// TIA Portal V19 export
FUNCTION_BLOCK "Pu_Versorgung.GP0x"   // FB1010, LAD
{ S7_Optimized_Access := 'TRUE' }
// Funktionen:  HF Versorgung  / Spülen
// stored: AutoNumber false, MemoryReserve 100, SetENOAutomatically false
   VAR RETAIN
      In { ExternalVisible := 'False'; ExternalWritable := 'False'} : Struct
         Auto : Bool;   // Paneltaste
         Ein : Bool;   // Paneltaste
         Not_Halt : Bool;
         Quitt_Al_Dfl : Bool;
         kein_Gas_Alarm : Bool;
         Leckage_Pumpe_ok : Bool;
         Leckage_PFA_Uebergang_ok : Bool;
         Leckage_Doppelrohr_ok : Bool;
         Leckage_Uml_Tunnel_ok : Bool;
         Leckage_Doppelschlauch_ok : Bool;
         Niv_min : Bool;
         Niv_max : Bool;
         Niv_Min_CM01 : Bool;
         Niv_Max_CM01 : Bool;
         Niv_Übervoll_CM01 : Bool;
         Niv_Min_CM02 : Bool;
         Niv_Max_CM02 : Bool;
         Niv_Übervoll_CM02 : Bool;
         Frg_Niv_CM05 : Bool;
         SRM_Saugseite_auf : Bool;
         SRM_Saugseite_zu : Bool;
         SRM_Druckseite_auf : Bool;
         SRM_Druckseite_zu : Bool;
         SRM_Eingang_Spülltg_auf : Bool;
         SRM_Eingang_Spülltg_zu : Bool;
         SRM_Ausgang_Spülltg_auf : Bool;
         SRM_Ausgang_Spülltg_zu : Bool;
         SRM_Versogung_UV01_auf : Bool;
         SRM_Versogung_UV01_zu : Bool;
         SRM_UV01_CM01_auf : Bool;
         SRM_UV01_CM01_zu { ExternalAccessible := 'False'} : Bool;
         SRM_UV01_CM02_auf { ExternalAccessible := 'False'} : Bool;
         SRM_UV01_CM02_zu { ExternalAccessible := 'False'} : Bool;
         Anf_HF_CM01 { ExternalAccessible := 'False'} : Bool;
         Anf_HF_CM02 { ExternalAccessible := 'False'} : Bool;
         IBC_vorhanden { ExternalAccessible := 'False'} : Bool;
         Tuer_vorn_zu { ExternalAccessible := 'False'} : Bool;
         Tuer_seitlich_zu { ExternalAccessible := 'False'} : Bool;
         Imp_Dfl { ExternalAccessible := 'False'} : Bool;
         GW_Dfl { ExternalAccessible := 'False'} : Bool;
         Betriebsart { ExternalAccessible := 'False'} : USInt := 0;   // Paneltaste
         Niveau { ExternalAccessible := 'False'} : USInt;
         Dfl { ExternalAccessible := 'False'} : Real;
      END_STRUCT;
      Param { ExternalAccessible := 'False'; ExternalVisible := 'False'; ExternalWritable := 'False'} : Struct
         Spülzeit : Time;
      END_STRUCT;
      Zst { ExternalAccessible := 'False'; ExternalVisible := 'False'; ExternalWritable := 'False'} : Struct
         Niveau : USInt;
         Status_GP0x : USInt;
         Restzeit_Spülen : Time;
         Spuelen : Bool;
         Pumpen : Bool;
         Weg_frei : Bool;
         Spuelen_aktiv : Bool;
         Bedienung_erlaubt : Bool;
      END_STRUCT;
      Mld { ExternalVisible := 'False'; ExternalWritable := 'False'} : Struct
         Leckage_Pumpe : Bool;
         Leckage_PFA_Uebergang : Bool;
         Leckage_Doppelrohr : Bool;
         Leckage_Uml_Tunnel : Bool;
         Leckage_Doppelschlauch : Bool;
         Niv_Sensorfehler : Bool;
         GW_Dfl : Bool;
         UeW_Dfl_Dos : Bool;
         Leermeldung : Bool;
         Vollmeldung : Bool;
         n_Auto : Bool;
         Radarsonde_niO : Bool;
      END_STRUCT;
      Out { ExternalVisible := 'False'; ExternalWritable := 'False'} : Struct
         GP0x_Ein : Bool;
         Spülventil_Eingang : Bool;
         Spülventil_Ausgang : Bool;
         Ventil_Saugseite : Bool;
         Ventil_Druckseite : Bool;
         Ventil_Entsorgung : Bool;
         Versorgung_UV01 : Bool;
         UV01_CM01 : Bool;
         UV01_CM02 : Bool;
      END_STRUCT;
   END_VAR
   VAR
      IEC_Timer : Struct
         GW_Dfl { ExternalAccessible := 'False'; ExternalVisible := 'False'; ExternalWritable := 'False'; S7_SetPoint := 'True'} : TON_TIME;
         Spülen { S7_SetPoint := 'True'} : TP_TIME;
         Verz_Min { S7_SetPoint := 'True'} : TON_TIME;
         Imp_Dfl { S7_SetPoint := 'True'} : TON_TIME;
         Spülventil_Ausgang { S7_SetPoint := 'True'} : TOF_TIME;
         Verz_NivMax { S7_SetPoint := 'True'} : TON_TIME;
      END_STRUCT;
      R_TRIG_Hand_EIN { S7_SetPoint := 'True'} : R_TRIG;
   END_VAR
   VAR_TEMP
      Spülzeit : Time;
      posFl_Hand : Bool;
      Leckage_Versorgung_ok : Bool;
      Alarm_Dfl_Dos : Bool;
   END_VAR
   VAR CONSTANT
      Niv_TLS : USInt := 2;
      Niv_Min : USInt := 20;
      Niv_max : USInt := 90;
      Zeit_Ventil_auf : Time := T#5s;
   END_VAR
BEGIN

REGION Network 1 (SCL): Input
   // Panelbedienung und Sensoren --> Input()

   // positive Flanke "Hand Ein"
   #R_TRIG_Hand_EIN(CLK := #In.Ein,
                    Q => #posFl_Hand);
   // Freigabe Not-Halt Pumpen
   #In.Not_Halt := NOT "DB_PNOZ_IN_Out".In.NH_Frg_Pumpen OR NOT "E_Frg_AbLW";

   // Leckage Versorgung
   #Leckage_Versorgung_ok := #In.Leckage_Doppelrohr_ok AND #In.Leckage_PFA_Uebergang_ok AND #In.Leckage_Uml_Tunnel_ok AND #In.Leckage_Doppelschlauch_ok;

   // Quittierung Alarm Durchfluss
   IF #In.Quitt_Al_Dfl AND #Mld.UeW_Dfl_Dos THEN
       #Mld.UeW_Dfl_Dos := FALSE;
   END_IF;
END_REGION

REGION Network 2 (SCL): Ansteuerung
   // Alles AUS
   IF (#In.Betriebsart = 3) AND #In.Tuer_vorn_zu AND #In.Tuer_seitlich_zu AND NOT #In.Not_Halt THEN // Spülen
       // Ausschaltverzögert - Druckabbau
       #IEC_Timer.Spülventil_Ausgang(IN := #Out.Spülventil_Eingang,
                                     PT := T#3s,
                                     Q => #Out.Spülventil_Ausgang);
   ELSE
       #Out.Spülventil_Eingang := FALSE;
       #Out.Spülventil_Ausgang := FALSE;
   END_IF;

   #Zst.Restzeit_Spülen := T#0s;
   #Out.Ventil_Saugseite := FALSE;
   #Out.Ventil_Druckseite := FALSE;
   #Out.Versorgung_UV01 := FALSE;
   #Out.UV01_CM01 := FALSE;
   #Out.UV01_CM02 := FALSE;
   #Out.Ventil_Entsorgung := FALSE;
   #Out.GP0x_Ein := FALSE;

   IF #In.Tuer_vorn_zu AND #In.Tuer_seitlich_zu AND NOT #In.Not_Halt THEN
       CASE #In.Betriebsart OF
           0:  // Versorgung Auto

               // Ventile öffnen
               IF #Leckage_Versorgung_ok AND #In.kein_Gas_Alarm THEN
                   #Out.Ventil_Saugseite := #Out.Ventil_Druckseite := #Out.Versorgung_UV01 := #In.Auto;
                   #Out.UV01_CM01 := #In.Anf_HF_CM01 AND #In.Auto;
                   #Out.UV01_CM02 := #In.Anf_HF_CM02 AND #In.Auto;
               END_IF;

               // Check weg
               #Zst.Weg_frei := #In.SRM_Ausgang_Spülltg_zu AND #In.SRM_Eingang_Spülltg_zu AND
               #In.SRM_Druckseite_auf AND #In.SRM_Saugseite_auf AND #In.SRM_Versogung_UV01_auf AND
               ((#In.SRM_UV01_CM01_auf AND #In.SRM_UV01_CM02_zu AND #In.Anf_HF_CM01) OR (#In.SRM_UV01_CM02_auf AND #In.SRM_UV01_CM01_zu AND #In.Anf_HF_CM02));

               // Weg frei, Behälter nicht leer und Ziel nicht übervoll
               #Zst.Pumpen := #Zst.Weg_frei AND NOT #Mld.Leermeldung AND #In.IBC_vorhanden AND NOT #Mld.UeW_Dfl_Dos AND
               ((#In.Anf_HF_CM01 AND NOT #In.Niv_Übervoll_CM01 AND NOT #In.Niv_Max_CM01) OR (#In.Anf_HF_CM02 AND NOT #In.Niv_Übervoll_CM02 AND NOT #In.Niv_Max_CM02));

           1:  // Versorgung CM01 Hand
               // Ventile öffnen
               IF #Leckage_Versorgung_ok AND #In.kein_Gas_Alarm THEN
                   #Out.Ventil_Saugseite := #Out.Ventil_Druckseite := #Out.Versorgung_UV01 := #Out.UV01_CM01 := #In.Ein;
               END_IF;

               // Check weg
               #Zst.Weg_frei := #In.SRM_Ausgang_Spülltg_zu AND #In.SRM_Eingang_Spülltg_zu AND
               #In.SRM_Druckseite_auf AND #In.SRM_Saugseite_auf AND
               #In.SRM_Versogung_UV01_auf AND #In.SRM_UV01_CM01_auf AND #In.SRM_UV01_CM02_zu;

               // Weg frei, Behälter nicht leer und Ziel nicht übervoll
               #Zst.Pumpen := #Zst.Weg_frei AND NOT #Mld.Leermeldung AND #In.IBC_vorhanden AND NOT #In.Niv_Übervoll_CM01 AND NOT #In.Niv_Max_CM01 AND NOT #In.Niv_Min_CM01;

           2:  // Versorgung CM02 Hand
               // Ventile öffnen
               IF #Leckage_Versorgung_ok AND #In.kein_Gas_Alarm THEN
                   #Out.Ventil_Saugseite := #Out.Ventil_Druckseite := #Out.Versorgung_UV01 := #Out.UV01_CM02 := #In.Ein;
               END_IF;

               // Check Weg
               #Zst.Weg_frei := #In.SRM_Ausgang_Spülltg_zu AND #In.SRM_Eingang_Spülltg_zu AND
               #In.SRM_Druckseite_auf AND #In.SRM_Saugseite_auf AND
               #In.SRM_Versogung_UV01_auf AND #In.SRM_UV01_CM02_auf AND #In.SRM_UV01_CM01_zu;

               // Weg frei, Behälter nicht leer und Ziel nicht übervoll
               #Zst.Pumpen := #Zst.Weg_frei AND NOT #Mld.Leermeldung AND #In.IBC_vorhanden AND NOT #In.Niv_Übervoll_CM02 AND NOT #In.Niv_Max_CM02 AND NOT #In.Niv_Min_CM02;

           3: // Spülen - nur Hand
               #Zst.Pumpen := FALSE;

               IF #In.Ein THEN
                   IF #posFl_Hand THEN
                       #Zst.Spuelen_aktiv := TRUE;
                   END_IF;
                   #Out.Spülventil_Eingang := #In.Frg_Niv_CM05 AND #In.SRM_Saugseite_zu AND #In.SRM_Druckseite_zu AND #Zst.Spuelen_aktiv;

                   #IEC_Timer.Spülen(IN := #In.SRM_Eingang_Spülltg_auf AND #In.SRM_Ausgang_Spülltg_auf,
                                     PT := #Param.Spülzeit,
                                     Q => #Zst.Spuelen,
                                     ET => #Spülzeit);
                   #Zst.Restzeit_Spülen := #Param.Spülzeit - #Spülzeit;

                   IF #In.SRM_Eingang_Spülltg_auf AND #In.SRM_Ausgang_Spülltg_auf AND #In.SRM_Saugseite_zu AND #In.SRM_Druckseite_zu
                       AND NOT #Zst.Spuelen AND #Zst.Spuelen_aktiv THEN
                       #Zst.Spuelen_aktiv := FALSE;
                       #Out.Spülventil_Eingang := FALSE;
                   END_IF;

               ELSE
                   #Out.Spülventil_Eingang := FALSE;
                   #Out.Spülventil_Ausgang := FALSE;
                   #Zst.Spuelen := FALSE;
                   #Zst.Spuelen_aktiv := FALSE;
               END_IF;

           4: // Entsorgung
               #Zst.Spuelen := FALSE;
               #Zst.Pumpen := FALSE;

               //Quick Connect Entsorgung
               #Out.Ventil_Entsorgung := NOT #In.Niv_max AND (#In.Niveau < 85) AND #In.IBC_vorhanden;

       END_CASE;
       // Pumpe an 
       #Out.GP0x_Ein := #Zst.Pumpen AND #In.Leckage_Pumpe_ok;
   END_IF;
END_REGION

REGION Network 3 (SCL): Überwachung / Meldungen
   // Durchflussüberwachung
   #IEC_Timer.Imp_Dfl(IN := NOT #In.Imp_Dfl AND #Zst.Pumpen AND (#In.Anf_HF_CM01 OR #In.Anf_HF_CM02),
                       PT := T#5s,
                       Q => #Alarm_Dfl_Dos);

    IF #Alarm_Dfl_Dos THEN
        #Mld.UeW_Dfl_Dos := TRUE;
    END_IF;

   // Meldungen Leckage 

   #Mld.Leckage_Pumpe := NOT #In.Leckage_Pumpe_ok;

   #Mld.Leckage_PFA_Uebergang := NOT #In.Leckage_PFA_Uebergang_ok;

   #Mld.Leckage_Doppelrohr := NOT #In.Leckage_Doppelrohr_ok;

   #Mld.Leckage_Uml_Tunnel := NOT #In.Leckage_Uml_Tunnel_ok;

   #Mld.Leckage_Doppelschlauch := NOT #In.Leckage_Doppelschlauch_ok;

   #IEC_Timer.GW_Dfl(IN := #In.GW_Dfl AND #Out.GP0x_Ein AND #In.SRM_Druckseite_auf,
                     PT := T#5s,
                     Q => #Mld.GW_Dfl);

   // Verzögerung Leermeldung
   #IEC_Timer.Verz_Min(IN := NOT #In.Niv_min AND #In.SRM_Saugseite_auf,
                       PT := T#5s,
                       Q => #Mld.Leermeldung);

   #Mld.Vollmeldung := #In.Niv_max AND (#In.Betriebsart = 4) AND #In.IBC_vorhanden;

   // nicht in Automatik
   #Mld.n_Auto := NOT #In.Auto AND "DB_ANLAGE".BA.Automat_ein AND #In.IBC_vorhanden;

   //Plausibiltät Radarsonde
   #Mld.Radarsonde_niO := ((#In.Niv_max AND (#In.Niveau < 85)) OR (NOT #In.Niv_max AND (#In.Niveau > 95)))
   AND #In.IBC_vorhanden;
END_REGION

REGION Network 4 (SCL): --> Visu
   // Status Pumpe
   "Status_E0A"(Hand := #In.Ein,
                Auto := #In.Auto,
                SonderModus_PumpeSpuelen:=FALSE,
                Stoerung := FALSE,
                Ausgang := #Out.GP0x_Ein,
                StatusByte => #Zst.Status_GP0x);
   // Anzeige Füllstand
   "Niv_Visu"(Niv_1 := #In.Niv_min,
              Niv_2 := #In.Niv_max,
              Niv_3 := FALSE,
              Niv_4 := FALSE,
              Niv_5 := FALSE,
              Niv_6 := FALSE,
              Wert_1 := #Niv_Min,
              Wert_2 := #Niv_max,
              Wert_3 := 0,
              Wert_4 := 0,
              Wert_5 := 0,
              Wert_6 := 0,
              Niveau => #Zst.Niveau,
              Niv_Err => #Mld.Niv_Sensorfehler);

   // Radarsonde
   #Zst.Niveau := #In.Niveau;
   #Zst.Bedienung_erlaubt := NOT #In.Ein AND NOT #In.Auto;
END_REGION
END_FUNCTION_BLOCK
